{attribute addProperty BoxType "AX5118-0000-0011-0011"}
{attribute addProperty Id "Master_control_wordAT %Q*UINT1620Velocity_command_valueAT %Q*DINT3240"}
{attribute addProperty CRC "1202223311"}
{attribute addProperty SizeInBites "48"}
{attribute addProperty SizeInBytes "6"}
TYPE MDT_47A878CF :
STRUCT
	{attribute addProperty Name "Master_control_word"}
	Master_control_word AT %Q* : UINT;
	{attribute addProperty Name "Velocity_command_value"}
	Velocity_command_value AT %Q* : DINT;
END_STRUCT
END_TYPE

(* stored: Version 1.2.0.0, ProductVersion 3.1.4024.9
   DUT MDT_47A878CF: Id {960ca583-23e2-44cd-8904-8684c94d2633} *)
